TYPE Decimal : LREAL; END_TYPE

(* stored: Version 1.1.0.1
   DUT Decimal: Id {1445bc49-7abe-4bdc-98cb-0563cc327d49} *)
